// TIA Portal project "PLC_Test" (V20)

(* hardware
DEVICE "ET 200SP station_1"  ET 200SP-Station
   slot 0: "Rack_0"  Rack  6ES5 710-8MAx1
   slot 1: "PLC_1"  CPU 1512SP F-1 PN  6ES7 512-1SK01-0AB0  V2.9
      slot 32768: "PROFINET interface_1"  X1
   slot 2: "Server module_1"  Server module  6ES7 193-6PA00-0AA0  V1.1
      slot 1: "Server module_1"  Server module
   slot 127: "BA 2xRJ45"  BA 2xRJ45  6ES7 193-6AR00-0AA0  V0.0
      slot 32769: "Port_1"  X1 P1  6ES7 193-6AR00-0AA0
      slot 32770: "Port_2"  X1 P2  6ES7 193-6AR00-0AA0
*)

// ===== PLC "PLC_1"  CPU 1512SP F-1 PN =====

VAR_GLOBAL   // PLC tag table "Default tag table"
   "Clock_Byte" AT %MB0 : Byte;
   "Clock_10Hz" AT %M0.0 : Bool;
   "Clock_5Hz" AT %M0.1 : Bool;
   "Clock_2.5Hz" AT %M0.2 : Bool;
   "Clock_2Hz" AT %M0.3 : Bool;
   "Clock_1.25Hz" AT %M0.4 : Bool;
   "Clock_1Hz" AT %M0.5 : Bool;
   "Clock_0.625Hz" AT %M0.6 : Bool;
   "Clock_0.5Hz" AT %M0.7 : Bool;
END_VAR

// folder: DataBlock

DATA_BLOCK "DB_Scambio_Dati"   // DB1
TITLE = DB di appoggio
{ S7_Optimized_Access := 'FALSE' }
AUTHOR : Nicola
VERSION : 0.1
// In questa DB vengono salvati i dati che saranno messi in comunicazione con l'applicazione esterna
   VAR
      "A" : Real := 1.0;   // DB1.DBD0 (4 Bytes)
      "B" : Real := -4.0;   // DB1.DBD4
      C : Real := 2.0;   // DB1.DBD8
      X_1 : Real;   // DB1.DBD12
      X_2 : Real;   // DB1.DBD16
      Msg : String;   // DB1.DBB20 (256 Bytes)
      Last_Cmd_Msg : String;
      Cmd_Solve : Bool;   // DB1.DBX256.0
      Cmd_Interrupt : Bool;
      Cmd_Continue : Bool;
      Cmd_Reset : Bool;
      Point : Struct   // Struttura punto
         X : Real;   // Coordinata X della struttura Point
         Y : Real;   // Coordinate Y della struttura Point
      END_STRUCT;
      Vel : Struct
         X : Real;
         Y : Real;
      END_STRUCT;
   END_VAR
BEGIN
END_DATA_BLOCK

// folder: Instances

DATA_BLOCK "Solver_DB"   // DB2
{ S7_Optimized_Access := 'TRUE' }
AUTHOR : Nicola
VERSION : 0.1
// stored: InstanceOfName Solver
"Solver"
BEGIN
END_DATA_BLOCK

// folder: (top level)

ORGANIZATION_BLOCK "Main"   // OB1, LAD, ProgramCycle
TITLE = "Main Program Sweep (Cycle)"
{ S7_Optimized_Access := 'TRUE' }
VERSION : 0.1
   VAR_INPUT
      Initial_Call : Bool;   // Initial call of this OB
      Remanence : Bool;   // =True, if remanent data are available
   END_VAR
BEGIN

REGION Network 1
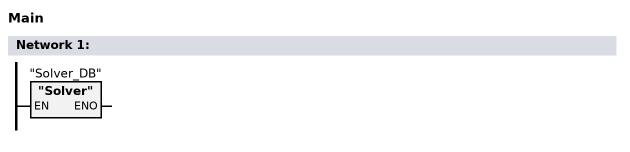
   RUNG wire#powerrail
      "Solver_DB"()
   END_RUNG
   // the same network as SCL:
   "Solver_DB"();   // "Solver"
END_REGION
END_ORGANIZATION_BLOCK

// folder: FunctionBlock

FUNCTION_BLOCK "Solver"   // FB1, SCL
TITLE = Gestione delle funzioni per soluzione equazioni
{ S7_Optimized_Access := 'TRUE' }
AUTHOR : Nicola
VERSION : 0.1
// In questa FB utilizzate le funzioni per soluzioni di equazioni
   VAR
      bOk : Bool;
      bContinue : Bool;
      bStartTimer : Bool;
      Sleep_timer_Instance : "Sleep_timer";
      Last_Cmd : Int;   // Indice associato all'ultimo comando chiamato
   END_VAR
   VAR_TEMP
      nX : Real;   // Step per il calcolo dei valori di ascissa
      tTimeSleep : Time;   // Tempo di attesa
      bNew_Cmd : Bool;   // Richiesta di esecuzione comando
   END_VAR
   VAR CONSTANT
      nStepX : Real := 0.1;
   END_VAR
BEGIN
   REGION COMMAND  
       // se richiesto di esguire il calolo: salvo i dati per averli già pronti al passo successvio
       IF "DB_Scambio_Dati".Cmd_Solve THEN
           // salvo il riferimento del comando che è stato eseguito
           #Last_Cmd := 1;
           // notifico che stato avviato un comando 
           #bNew_Cmd := TRUE;
           // salvo nella variabile locale STATICA che l'operazione è andata a buon fine
           #bOk := FALSE;
           // Procedo al calcolo degli zeri
           IF "Solver_Quadratic_Eq"(a := "DB_Scambio_Dati".A, b := "DB_Scambio_Dati".B, c := "DB_Scambio_Dati".C,
                                        x_1 => "DB_Scambio_Dati".X_1,
                                        x_2 => "DB_Scambio_Dati".X_2) THEN
               // operazione riuscita
               "DB_Scambio_Dati".Msg := 'Equazione secondo grado risolta';
               // salvo nella variabile locale che l'operazione è andata a buon fine
               #bOk := TRUE;
               // Salvo il primo il punto dell'intervallo (x_1 è per definizione minore di x_2)
               "DB_Scambio_Dati".Point.X := "DB_Scambio_Dati".X_1;
           ELSIF "DB_Scambio_Dati".A = 0 THEN
               // Procedo al colcolo degli zeri     
               IF "Solver_Linera_Eq"(b := "DB_Scambio_Dati".B, c := "DB_Scambio_Dati".C,
                                         x_1 => "DB_Scambio_Dati".X_1) THEN
                   "DB_Scambio_Dati".Msg := 'Equazione primo grado';
               END_IF;
           ELSE
               // operazione non riuscita in campo reale
               "DB_Scambio_Dati".Msg := 'Equazione secondo grado non risolvibile in campo reale';
           END_IF;
           // al termine dell'esecuzione del comando resetto la variabile
           "DB_Scambio_Dati".Cmd_Solve := False;
       END_IF;

       // Se chiesto Reset interrimpo tutte le operazioni
       IF "DB_Scambio_Dati".Cmd_Interrupt THEN
           // salvo il riferimento del comando che è stato eseguito
           #Last_Cmd := 2;
           // notifico che stato avviato un comando 
           #bNew_Cmd := TRUE;
           // tutti i punti sono stati restituiti, quindi interrompo
           #bOk := False;
           // avviso che sono stati processati tutti i valori
           "DB_Scambio_Dati".Msg := 'Forzata interruzione';
           // Resetto la variabile
           "DB_Scambio_Dati".Cmd_Interrupt := FALSE;
       END_IF;

       // Se chiesto riavvio del ciclo di calcolo dei punti
       IF "DB_Scambio_Dati".Cmd_Continue THEN
           // salvo il riferimento del comando che è stato eseguito
           #Last_Cmd := 3;
           // notifico che stato avviato un comando 
           #bNew_Cmd := TRUE;
           // riavvio il ciclo (la funzione che restituisce i punti verificherà se procedere)
           #bOk := TRUE;
           // avviso che sono stati processati tutti i valori
           "DB_Scambio_Dati".Msg := 'Forzato riavvio';
           // Resetto la variabile
           "DB_Scambio_Dati".Cmd_Continue := FALSE;
       END_IF;

       IF "DB_Scambio_Dati".Cmd_Reset THEN
           // salvo il riferimento del comando che è stato eseguito
           #Last_Cmd := 4;
           // notifico che stato avviato un comando 
           #bNew_Cmd := TRUE;
           // interrompo il ciclo
           #bOk := FALSE;
           // avviso che sono stati processati tutti i valori
           "DB_Scambio_Dati".Msg := 'Forzato reset';
           // Azzero i dati iniziali di calcolo
           "DB_Scambio_Dati".Point.X := 0.0;
           "DB_Scambio_Dati".Point.Y := 0.0;
           "DB_Scambio_Dati".Vel.X := 0.0;
           "DB_Scambio_Dati".Vel.Y := 0.0;
           // Resetto la variabile
           "DB_Scambio_Dati".Cmd_Reset := FALSE;
       END_IF;

   END_REGION Command

   REGION METHODS   
       // se l'equazione è stata risolta allora procedo a restituire le coppie di valori (x,y) nell'intervallo degli zeri
       IF #bOk AND "DB_Scambio_Dati".Point.X <= "DB_Scambio_Dati".X_2 THEN
           // Ogni T secondi genero un impulso che fa eseguire l'operazione che segue
           #Sleep_timer_Instance(tTime_Sleep := t#2s);
           IF #Sleep_timer_Instance.bTime_Out THEN
               // determino la nuova coordinata X del punto
               "DB_Scambio_Dati".Point.X := "DB_Scambio_Dati".Point.X + #nStepX;
               // se il punto è dentro l'intervallo allora procedo al calcolo
               IF "DB_Scambio_Dati".Point.X <= "DB_Scambio_Dati".X_2 THEN
                   // Procedo a fare il calcolo del valore
                   "Value_of_Quadratic_Eq"(a := "DB_Scambio_Dati".A,
                                           b := "DB_Scambio_Dati".B,
                                           c := "DB_Scambio_Dati".C,
                                           Point := "DB_Scambio_Dati".Point,
                                           Vel := "DB_Scambio_Dati".Vel);
               ELSE
                   // tutti i punti sono stati restituiti, quindi interrompo
                   #bOk := False;
                   // avviso che sono stati processati tutti i valori
                   "DB_Scambio_Dati".Msg := 'Terminato valori';
               END_IF;
           END_IF;

       END_IF;

       // Se è stato lanciato un nuovo comando allora cerco il messaggio associato
       IF #bNew_Cmd THEN
           // Asseganto l'indice del comando restituisce il suo messaggio
           "DB_Scambio_Dati".Last_Cmd_Msg := "Get_Msg_From_Ind"(Ind_Cmd := #Last_Cmd);
           // per sicurezza resetto lo stato 
           #bNew_Cmd := FALSE;
       END_IF;

   END_REGION Methods
END_FUNCTION_BLOCK

FUNCTION_BLOCK "Sleep_timer"   // FB2, SCL
TITLE = Ogni Ts genera impulso in uscita
{ S7_Optimized_Access := 'TRUE' }
AUTHOR : Nicola
VERSION : 0.1
// Riceve in ingresso il tempo Ts e il bit di attivazione, per tutto il tempo chela FB è attiva viene generato un impulso in uscita ogni Ts+1TempoCiclo (il tempo ciclo che viene sommato è immpiegato per eseguire il reset del timer)
   VAR_INPUT
      tTime_Sleep : Time;
   END_VAR
   VAR_OUTPUT
      bTime_Out : Bool;   // Booleano che identifica il raggiungimento del tempo
   END_VAR
   VAR
      ms_Delay_Timer : TON_TIME;
      ms_bStartTimer : Bool;
      ms_bContinue : Bool;
   END_VAR
   VAR_TEMP
      mt_tTimeSleep : Time;
   END_VAR
BEGIN
   // Se è stato generato l'impulso
   IF #ms_bContinue THEN
       // Resetto la variabile per poter generare il fronte di salita
       #ms_bStartTimer := FALSE;
       #bTime_Out := FALSE;
   ELSIF NOT #ms_bContinue AND NOT #ms_bStartTimer THEN
       // Setto la variabile per lo start del timer
       #ms_bStartTimer := TRUE;
   END_IF;
   // Avvio il timer
   #ms_Delay_Timer(IN := #ms_bStartTimer, PT := #tTime_Sleep, Q => #ms_bContinue, ET => #mt_tTimeSleep);
   IF #ms_Delay_Timer.Q THEN
       // Resetto le variabili di questa FB
       #mt_tTimeSleep := t#0s;
       #bTime_Out := TRUE;
   END_IF;
END_FUNCTION_BLOCK

// folder: Functions

FUNCTION "Solver_Quadratic_Eq" : Bool   // FC1, SCL
TITLE = Ricerca degli zeri di un'equazione di secondo grado
{ S7_Optimized_Access := 'TRUE' }
AUTHOR : Nicola
VERSION : 0.1
// Inseriti i parametri a,b,c di un'equazione di secondo grado espressa nella forma esplicita "a*x^2 + b*x + c = 0" restituisce le soluzioni (se esistono)
   VAR_INPUT
      "a" : Real;   // Coefficiente associato a "x^2"
      "b" : Real;   // Coefficiente associato a "x"
      c : Real;   // Termine noto
   END_VAR
   VAR_OUTPUT
      x_1 : Real;   // Primo zero della funzione
      x_2 : Real;   // Secondo zero della funzione
   END_VAR
   VAR_TEMP
      delta : Real;
   END_VAR
BEGIN
   IF #a = 0 THEN
       #Solver_Quadratic_Eq := FALSE;
       RETURN;
   END_IF;
   // determino il valore del Delta al quadrato
   #delta := #b*#b - 4*#a*#c;
   // se il delta è maggiore di zero allora esista la soluzione nel campo reale
   IF #delta >= 0 THEN
       #delta := SQRT(#delta);
       #x_1 := (- #b - #delta) / (2 * #a);
       #x_2 := (- #b + #delta) / (2 * #a);
       // restituisco che l'operazione è andata a buon fine
       #Solver_Quadratic_Eq := TRUE;
   ELSE
       // restituisco che l'operazione è andata a buon fine
       #Solver_Quadratic_Eq := FALSE;
   END_IF;
END_FUNCTION

FUNCTION "Value_of_Quadratic_Eq" : Void   // FC2, SCL
TITLE = Restituisce il valore Y dell'equazione di secondo grado
{ S7_Optimized_Access := 'TRUE' }
AUTHOR : Nicola
VERSION : 0.1
// Fissati i parametri a, b, c dell'equazione di secondo grado in forma esplicita per il valore X in ingresso restitcuisce il valore f(X) e f'(x)
   VAR_INPUT
      "a" : Real;   // Coefficiente associato a "x^2"
      "b" : Real;   // Coefficiente associato a "x"
      c : Real;   // Termine noto
   END_VAR
   VAR_IN_OUT
      Point : Struct
         X : Real;
         Y : Real;
      END_STRUCT;
      Vel : Struct
         X : Real;
         Y : Real;
      END_STRUCT;
   END_VAR
BEGIN
   // Determino il valore puntuale dell'equazione di secondo grado
   #Point.Y := #a * #Point.X * #Point.X + #b * #Point.X + #c;
   // Definisco il valore x della derivata
   #Vel.X := #Point.X;
   // Determino il valore puntuale della derivata
   #Vel.Y := 2*#a*#Vel.X + #b;
END_FUNCTION

FUNCTION "Solver_Linera_Eq" : Bool   // FC3, SCL
TITLE = Solutore di equazione di primo grado
{ S7_Optimized_Access := 'TRUE' }
AUTHOR : Nicola
VERSION : 0.1
// Assegnata l'equazione lineare nella forme b*x + c = 0 restituisce lo zero dell'eqauzione.
   VAR_INPUT
      "b" : Real;   // Coefficiente associato a "x"
      c : Real;   // Termine noto
   END_VAR
   VAR_OUTPUT
      x_1 : Real;   // Zero della funzione
   END_VAR
BEGIN
   // se non è un'equazione lineare ritorno falso
   IF #b = 0 THEN
       #Solver_Linera_Eq := FALSE;
       RETURN;
   END_IF;
   // Prcedo alla ricerca dello zero dell'equazione
   #x_1 := - #c / #b;
   #Solver_Linera_Eq := TRUE;
END_FUNCTION

FUNCTION "Get_Msg_From_Ind" : String   // FC4, SCL
TITLE = Restituisce il messaggio associato all'indice
{ S7_Optimized_Access := 'TRUE' }
AUTHOR : Nicola Pievani
VERSION : 0.1
// In funzione dell'indice che il metodo riceve viene restituito il messaggio associato
   VAR_INPUT
      Ind_Cmd : Int;   // Indice del comando
   END_VAR
   VAR_TEMP
      Msg_Cmd : String;
   END_VAR
BEGIN
   // Recupera il messaggio associato all'indice (la definizione dell'indice del comando è definito nella FB1)
   CASE #Ind_Cmd OF
       1:
           #Msg_Cmd := 'Solve';
       2:
           #Msg_Cmd := 'Interrupt';
       3:
           #Msg_Cmd := 'Continue';
       4:
           #Msg_Cmd := 'Reset';
       ELSE
           #Msg_Cmd := ' --- ';
   END_CASE;
   // Restituisce il messaggio
   #Get_Msg_From_Ind := #Msg_Cmd;
END_FUNCTION